// TIA Portal V19 export
TYPE "dtStageUp"
   STRUCT
      zoneChangeOP : Real := 95.0;
      delayUpgrade { S7_SetPoint := 'True'} : Time := T#5S;
   END_STRUCT;
END_TYPE
